# B&R Automation Studio project mpdata
Automation Studio 4.2.12.129 SP; Default project; technology packages: mapp 1.66.0, TextSystem 

## Configuration Simulation

CPU , AutomationRuntime G4.26

### Task classes (Cpu.sw)
```
Cyclic#1 (cycle 100000 us, tolerance 10000000 us):
  prog1 <- prog1.prg
Binaries: ashwd, arconfig, iomap, asfw, sysconf, Config
Libraries: AsIecCon, astime, MpData, DataObj, MpCom, sys_lib, brsystem, FileIO, Runtime, AsBrStr, standard, MpWebXs, AsArSdm, arsvcreg, IecCheck, MpBase
```

### Hardware
```
PC_any : PC_any v1.1.0.0 (OrderNumber=PC)
  ConfigurationID = mpdata_Simulation
  Cyclic1Duration = 100000
  Cyclic1Tolerance = 10000000
  Cyclic2Duration = 200000
  Cyclic2Tolerance = 10000000
  Cyclic3Duration = 500000
  Cyclic3Tolerance = 10000000
  Cyclic4Duration = 1000000
  Cyclic4Tolerance = 10000000
  Cyclic5Duration = 2000000
  Cyclic5Tolerance = 10000000
  Cyclic6Duration = 3000000
  Cyclic6Tolerance = 12000000
  Cyclic7Duration = 4000000
  Cyclic7Tolerance = 12000000
  Cyclic8Duration = 5000000
  Cyclic8Tolerance = 30000000
  FileDevice1
  FileDeviceName1 = hdd
  FileDevicePath1 = C:\temp
```

## Logical view

Binary libraries used (declarations not repeated): Runtime, Operator, AsIecCon, astime, DataObj, sys_lib, brsystem, FileIO, AsBrStr, standard, AsArSdm, MpCom 1.66.0, MpBase 5.03.0, MpData 1.66.0, MpWebXs 1.66.0

### Package Logical/Libraries - Global libraries

### Library Logical/Libraries/IecCheck (IEC)
Depends on: sys_lib, AsBrStr

#### IecCheck.fun - Exported functions and function blocks
```iecst
FUNCTION CheckDivDWord : UDINT (* Check divisor for DINT and UDINT division *)
	VAR_INPUT
		divisor : UDINT;
	END_VAR
END_FUNCTION

FUNCTION CheckDivWord : UINT (* Check divisor for INT and UINT division *)
	VAR_INPUT
		divisor : UINT;
	END_VAR
END_FUNCTION

FUNCTION CheckDivByte : USINT (* Check divisor for SINT and USINT division *)
	VAR_INPUT
		divisor : USINT;
	END_VAR
END_FUNCTION

FUNCTION CheckDivReal : REAL (* Check divisor for REAL division *)
	VAR_INPUT
		divisor : REAL;
	END_VAR
END_FUNCTION

FUNCTION CheckDivLReal : LREAL (* Check divisor for LREAL division, not available for SG3 and SGC *)
	VAR_INPUT
		divisor : LREAL;
	END_VAR
END_FUNCTION

FUNCTION CheckBounds : DINT (* Check range for array access *)
	VAR_INPUT
		index : DINT;
		lower : DINT;
		upper : DINT;
	END_VAR
END_FUNCTION

FUNCTION CheckRange : DINT (* Check range for enumeration *)
	VAR_INPUT
		value : DINT;
		lower : DINT;
		upper : DINT;
	END_VAR
END_FUNCTION

FUNCTION CheckSignedSubrange : DINT (* Check range for subrange of signed data types *)
	VAR_INPUT
		value : DINT;
		lower : DINT;
		upper : DINT;
	END_VAR
END_FUNCTION

FUNCTION CheckUnsignedSubrange : UDINT (* Check range for subrange of unsigned data types *)
	VAR_INPUT
		value : UDINT;
		lower : UDINT;
		upper : UDINT;
	END_VAR
END_FUNCTION

FUNCTION CheckReadAccess : UDINT (* Check address when reading dynamic variables *)
	VAR_INPUT
		address : UDINT;
	END_VAR
END_FUNCTION

FUNCTION CheckWriteAccess : UDINT (* Check address when writing dynamic variables *)
	VAR_INPUT
		address : UDINT;
	END_VAR
END_FUNCTION

FUNCTION MakeEntry : UDINT (* Makes an entry (log book entry) in the error log book *)
	VAR
		taskname : STRING[30];
		group : USINT;
		status_name : UINT;
		out_text : STRING[80];
	END_VAR
	VAR_INPUT
		number : UINT;
		index : DINT;
		text : STRING[50];
	END_VAR
END_FUNCTION
```

#### IecCheck.st - Implementation file
```iecst
(* Check divisor for DINT and UDINT division *)
FUNCTION CheckDivDWord
	IF divisor=0 THEN
		CheckDivDWord:=1;
		MakeEntry(55555,divisor,'CheckDivDWord');
	ELSE
		CheckDivDWord:=divisor;
	END_IF
END_FUNCTION

(* Check divisor for INT and UINT division *)
FUNCTION CheckDivWord
	IF divisor=0 THEN
		CheckDivWord:=1;
		MakeEntry(55555,divisor,'CheckDivWord');
	ELSE
		CheckDivWord:=divisor;
	END_IF
END_FUNCTION

(* Check divisor for SINT and USINT division *)
FUNCTION CheckDivByte
	IF divisor=0 THEN
		CheckDivByte:=1;
		MakeEntry(55555,divisor,'CheckDivByte');
	ELSE
		CheckDivByte:=divisor;
	END_IF
END_FUNCTION

(* Check divisor for REAL division *)
FUNCTION CheckDivReal
	IF divisor=0 THEN
		CheckDivReal:=1;
		MakeEntry(55555,0,'CheckDivReal');
	ELSE
		CheckDivReal:=divisor;
	END_IF
END_FUNCTION

(* Check divisor for LREAL division *)
FUNCTION CheckDivLReal
	IF divisor=0 THEN
		CheckDivLReal:=1;
		MakeEntry(55555,0,'CheckDivLReal');
	ELSE
		CheckDivLReal:=divisor;
	END_IF
END_FUNCTION

(* Check range for array access *)
FUNCTION CheckBounds
	IF index < lower THEN
		CheckBounds := lower;
		MakeEntry(55555,index,'CheckBounds');
	ELSIF index > upper THEN
		CheckBounds := upper;
		MakeEntry(55555,index,'CheckBounds');
	ELSE
		CheckBounds := index;
	END_IF
END_FUNCTION

(* Check range for enumeration *)
FUNCTION CheckRange
	IF value < lower THEN
		CheckRange := lower;
		MakeEntry(55555,value,'CheckRange');
	ELSIF value > upper THEN
		CheckRange := upper;
		MakeEntry(55555,value,'CheckRange');
	ELSE
		CheckRange := value;
	END_IF
END_FUNCTION

(* Check range for subrange of signed data types *)
FUNCTION CheckSignedSubrange
	IF value < lower THEN
		CheckSignedSubrange := lower;
		MakeEntry(55555,value,'CheckSignedSubrange');
	ELSIF value > upper THEN
		CheckSignedSubrange := upper;
		MakeEntry(55555,value,'CheckSignedSubrange');
	ELSE
		CheckSignedSubrange := value;
	END_IF
END_FUNCTION

(* Check range for subrange of unsigned data types *)
FUNCTION CheckUnsignedSubrange
	IF value < lower THEN
		CheckUnsignedSubrange := lower;
		MakeEntry(55555,value,'CheckUnsignedSubrange');
	ELSIF value > upper THEN
		CheckUnsignedSubrange := upper;
		MakeEntry(55555,value,'CheckUnsignedSubrange');
	ELSE
		CheckUnsignedSubrange := value;
	END_IF
END_FUNCTION

(* Check address when reading dynamic variables *)
FUNCTION CheckReadAccess
	IF address=0 THEN
		(* TODO: Insert an appropriate code, see AutomationStudio help for further information *)
		MakeEntry(55555,address,'Read from NULL');
	END_IF

	CheckReadAccess:=0;
END_FUNCTION

(* Check address when writing dynamic variables *)
FUNCTION CheckWriteAccess
	IF address=0 THEN
		(* TODO: Insert an appropriate code, see AutomationStudio help for further information *)
		MakeEntry(55555,address,'Write to NULL');
	END_IF

	CheckWriteAccess:=0;
END_FUNCTION

(* Makes an entry (log book entry) in the error log book *)
FUNCTION MakeEntry
		status_name := ST_name(0,ADR(taskname),ADR(group));

		brsstrcpy(ADR(out_text),ADR(text));
		brsstrcat(ADR(out_text),ADR(' > in task > '));
  		brsstrcat(ADR(out_text),ADR(taskname));
		MakeEntry := ADR(out_text);
		ERRxfatal(number,index,ADR(out_text));
END_FUNCTION
```

### Program Logical/prog1 (IEC)

#### Cyclic.st - Cyclic code
```iecst
PROGRAM _CYCLIC

	CASE step OF
	    0:  (* start data recorder *)
			MpDataRecorder_0.Enable := 1;
			IF( MpDataRecorder_0.Active )THEN
				step := 10;
			END_IF

		10: (* create columns and register variables *)
			MpDataRegPar_0(	Enable := 1 );
			MpDataRegPar_1(	Enable := 1 );
			MpDataRegPar_2(	Enable := 1 );

			IF(    (MpDataRegPar_0.Active = FALSE AND MpDataRegPar_0.Error = FALSE) AND
					(MpDataRegPar_1.Active = FALSE AND MpDataRegPar_1.Error = FALSE) AND
					(MpDataRegPar_2.Active = FALSE AND MpDataRegPar_2.Error = FALSE) ) THEN
				step := 100;
			END_IF

		100:  (* wait for command *)
		IF( writeCSV = 1) THEN
			writeCSV := 2; (* busy *)
			MpDataRecorder_0.Record := TRUE;
			index := 0;
			step := 200;
		END_IF

		200: (* next record *)
		IF( MpDataRecorder_0.Error ) THEN
			step := 900;  (* Fehler *)
		ELSE
			MpDataRecorder_0( Trigger := FALSE );
			record := data[index];
			index := index + 1;
			MpDataRecorder_0.Trigger := TRUE;
			IF ( index > (MAX_ROWS-1) ) THEN
				MpDataRecorder_0.Record := FALSE;
				writeCSV := 0;
				step := 100; (* ready *)
			END_IF
		END_IF

	END_CASE

	MpDataRecorder_0();

END_PROGRAM
```

#### Init.st - Init code
```iecst
PROGRAM _INIT

	(* simulation data *)
	FOR i:= 0 TO (MAX_ROWS-1) DO
		data[i].count := INT_TO_USINT(i+1);
		brsitoa( i+1, ADR(s1) );
		s2 := 'parameter ';
		s2 := CONCAT( s2, s1 );
		data[i].parameter := s2;
		data[i].value := 3.14 * i;
	END_FOR

	MpDataRecorder_0(	MpLink := ADR(gDataRecorder) ,
						Enable := 0,
						DeviceName := ADR('hdd'),
						RecordMode := mpDATA_RECORD_MODE_TRIGGER  );

	MpDataRegPar_0(		MpLink := ADR(gDataRecorder),
						Enable := 0,
						PVName := ADR('prog1:record.count'),
						Unit := ADR('St'),
						Description := ADR('count'),
						ScaleFactor := 1);

	MpDataRegPar_1(		MpLink := ADR(gDataRecorder),
						Enable := 0,
						PVName := ADR('prog1:record.parameter'),
						Unit := ADR('parameter'),
						Description := 0,
						ScaleFactor := 1);

	MpDataRegPar_2(		MpLink := ADR(gDataRecorder),
						Enable := 0,
						PVName := ADR('prog1:record.value'),
						Unit := ADR('value'),
						Description := 0,
						ScaleFactor := 1);

	step := 0;

END_PROGRAM
```

#### Types.typ - Local data types
```iecst
TYPE
	DataRecordTyp : 	STRUCT
		count : USINT;
		parameter : STRING[80];
		value : LREAL;
	END_STRUCT;
END_TYPE
```

#### Variables.var - Local variables
```iecst
VAR CONSTANT
	MAX_ROWS : UINT := 100;
END_VAR
VAR
	i : INT;
	index : UINT := 0;
	record : DataRecordTyp;
	data : ARRAY[0..MAX_ROWS] OF DataRecordTyp;
	s1 : STRING[80];
	s2 : STRING[80];
	step : UINT;
	MpDataRegPar_1 : MpDataRegPar;
	MpDataRegPar_2 : MpDataRegPar;
	MpDataRegPar_0 : MpDataRegPar;
	MpDataRecorder_0 : MpDataRecorder;
	writeCSV : USINT; (*Kommando*)
END_VAR
```

Listed in the project but not available here: Logical/Global.typ, Logical/Global.var, Logical/prog1/Exit.st
